(* IEC 61131-3 sources: test/Class/HmiComPortCan, 1 file *)

(* ---- HmiComPortCan.st ---- *)
(*!
<Class
	Name               = "HmiComPortCan"
	Revision           = "0.14"
	RealtimeTask       = "false"
	CyclicTask         = "false"
	BackgroundTask     = "false"
	Sigmatek           = "true"
	OSInterface        = "false"
	HighPriority       = "false"
	Automatic          = "false"
	UpdateMode         = "Prescan"
	SharedCommandTable = "true"
	Objectsize         = "(490,120)">
	<Channels>
		<Client Name="CanInterface" Required="true" Internal="false" DefValue="1"/>
		<Client Name="CanNodeDisplay" Required="true" Internal="false" DefValue="1"/>
		<Client Name="CanRxMsgID" Required="true" Internal="false" DefValue="16#40"/>
		<Client Name="CanSend" Required="true" Internal="true"/>
		<Client Name="CanTxMsgID" Required="true" Internal="false" DefValue="16#20"/>
		<Client Name="CoCanLib" Required="false" Internal="false"/>
	</Channels>
	<RevDoku>
		<Owner Company="sigmatek" Author="kolott"/>
		<Dokumentation Revision="0.14" Date="2015-06-11" Author="hoechr1" Company="sigmatek" Description="SA31241: inserted client for communication over hardware modules"/>
		<Dokumentation Revision="0.13" Date="2015-03-16" Author="kolott" Company="sigmatek" Description="SA30531: new Clients CanRxMsgID and CanTxMsgID"/>
		<Dokumentation Revision="0.12" Date="2014-11-27" Author="kolott" Company="sigmatek" Description="code reduced to can-connection"/>
		<Dokumentation Revision="0.11" Date="2014-08-28" Author="kolott" Company="sigmatek" Description="function &quot;UserCall&quot; added, extended timeout at flashkill &#13;&#10;retry implemented at method SendFile()"/>
		<Dokumentation Revision="0.10" Date="2014-06-13" Author="kolott" Company="sigmatek" Description="attribut &quot;virtual global&quot; added to method SendData()"/>
		<Dokumentation Revision="0.9" Date="2014-05-14" Author="kolott" Company="sigmatek" Description="evaluate retcode of method UpdateData()"/>
		<Dokumentation Revision="0.8" Date="2014-04-24" Author="kolott" Company="sigmatek" Description="new Method SendRestartSetup()"/>
		<Dokumentation Revision="0.7" Date="2014-04-02" Author="kolott" Company="sigmatek" Description="ErrorCnt will count on tx error as well"/>
		<Dokumentation Revision="0.6" Date="2014-03-04" Author="kolott" Company="sigmatek" Description="new Method GetNode()"/>
		<Dokumentation Revision="0.5" Date="2014-02-21" Author="kolott" Company="sigmatek" Description="new Method: GetHwVersion(), GetSwVersion()"/>
		<Dokumentation Revision="0.4" Date="2014-02-13" Author="kolott" Company="sigmatek" Description="innovation"/>
		<Dokumentation Revision="0.3" Date="2014-02-12" Author="kolott" Company="sigmatek" Description="new command LastUsage of HMI implemented"/>
		<Dokumentation Revision="0.2" Date="2014-01-29" Author="kolott" Company="sigmatek" Description="innovation: speed"/>
		<Dokumentation Revision="0.1" Date="2014-01-16" Author="kolott" Company="sigmatek" Description="method SendTrendValue added"/>
	</RevDoku>
	<Network Name="HmiComPortCan">
		<!-- List of Components in this network -->
		<Components>
			<Object
				Name       = "_base"
				Class      = "HmiComPort"
				Position   = "(218,120)"
				Visualized = "false">
				<Channels>
					<Server Name="ClassSvr"/>
					<Server Name="ErrorCnt"/>
					<Server Name="RetryCnt"/>
					<Server Name="RxData"/>
					<Server Name="TxData"/>
					<Client Name="CoSys"/>
					<Client Name="StdLib"/>
				</Channels>
			</Object>
			<Object
				Name       = "CanSend"
				Class      = "HmiCanSendReceive"
				Position   = "(210,510)"
				Visualized = "false">
				<Channels>
					<Server Name="ClassSvr"/>
					<Server Name="ErrorCnt"/>
					<Server Name="RxPack"/>
					<Server Name="TxPack"/>
					<Server Name="TxRetry"/>
					<Client Name="CanInterface" Value="1"/>
					<Client Name="CanNodeDisplay" Value="1"/>
					<Client Name="CanRxMsgID" Value="16#40"/>
					<Client Name="CanTxMsgID" Value="16#20"/>
					<Client Name="CoCan"/>
					<Client Name="CoCanLib"/>
					<Client Name="CoSys"/>
				</Channels>
			</Object>
		</Components>
		<Comments>
		</Comments>
		<!-- List of Connections in this network -->
		<Connections>
			<Connection Source="this.ClassSvr" Destination="_base.ClassSvr" Vertices="(690,210),(518,210),"/>
			<Connection Source="this.CanSend" Destination="CanSend.ClassSvr"/>
			<Connection Source="CanSend.CanNodeDisplay" Destination="this.CanNodeDisplay" Vertices="(210,600),(38,510),"/>
			<Connection Source="CanSend.CanInterface" Destination="this.CanInterface" Vertices="(210,660),(38,570),"/>
			<Connection Source="this.RxData" Destination="_base.RxData" Vertices="(690,270),(518,270),"/>
			<Connection Source="this.TxData" Destination="_base.TxData" Vertices="(690,330),(518,330),"/>
			<Connection Source="this.ErrorCnt" Destination="_base.ErrorCnt" Vertices="(690,390),(518,390),"/>
			<Connection Source="this.RetryCnt" Destination="_base.RetryCnt" Vertices="(690,450),(518,450),"/>
			<Connection Source="CanSend.CanRxMsgID" Destination="this.CanRxMsgID" Vertices="(210,720),(38,630),"/>
			<Connection Source="CanSend.CanTxMsgID" Destination="this.CanTxMsgID" Vertices="(210,780),(38,690),"/>
			<Connection Source="CanSend.CoCanLib" Destination="this.CoCanLib" Vertices="(210,960),(38,750),"/>
		</Connections>
		<!-- Headerfiles -->
		<Options>
		</Options>
	</Network>
</Class>
*)
#pragma using HmiComPort

HmiComPortCan : CLASS
: HmiComPort
  //Servers:
  //Clients:
	CanNodeDisplay 	: CltCh_DINT;
	CanInterface 	: CltCh_DINT;
	CanSend 	: CltChCmd_HmiCanSendReceive;
	CanRxMsgID 	: CltCh_DINT;
	CanTxMsgID 	: CltCh_DINT;
	CoCanLib 	: CltChCmd__CanLib;
  //Variables:
		RxCrc 	: UDINT;
		Crc 	: UDINT;
  //Functions:

	FUNCTION VIRTUAL GLOBAL Start
		VAR_INPUT
			pthis 	: ^void;
		END_VAR;

	FUNCTION VIRTUAL GLOBAL GetNode
		VAR_OUTPUT
			retcode 	: UDINT;
		END_VAR;

	FUNCTION VIRTUAL SendDataIntern
		VAR_INPUT
			src 	: ^void;
			size 	: UDINT;
		END_VAR
		VAR_OUTPUT
			retcode 	: BOOL;
		END_VAR;
				//! <Function Comment="Get timeout in milliseconds to wait for rx-data" Name="GetRxTimeout"/>
	FUNCTION VIRTUAL GetRxTimeout
		VAR_INPUT
			index 	: TRxTimeout;
		END_VAR
		VAR_OUTPUT
			retcode 	: UDINT;
		END_VAR;

	FUNCTION GLOBAL RxCallback
		VAR_INPUT
			pthis 	: ^HmiComPortCan;
			pdata 	: ^USINT;
			size 	: UDINT;
		END_VAR;
  //Tables:
	FUNCTION @STD
		VAR_OUTPUT
			ret_code	: CONFSTATES;
		END_VAR;
	FUNCTION GLOBAL TAB @CT_;
END_CLASS;

#pragma using HmiCanSendReceive
#pragma usingLtd _CanLib

FUNCTION VIRTUAL GLOBAL HmiComPortCan::Start
	VAR_INPUT
		pthis 	: ^void;
	END_VAR

  HmiComPort::Start(pthis);
  CanSend.Start(#RxCallback(), this);
  RetryNo := 2;  // 2 retry after first fail

END_FUNCTION

FUNCTION GLOBAL HmiComPortCan::RxCallback
	VAR_INPUT
		pthis 	: ^HmiComPortCan;
		pdata 	: ^USINT;
		size 	: UDINT;
	END_VAR

  this := pthis;
  RecieveData(pdata, size);

END_FUNCTION

FUNCTION VIRTUAL GLOBAL HmiComPortCan::GetNode
	VAR_OUTPUT
		retcode 	: UDINT;
	END_VAR

  retcode := to_udint(CanNodeDisplay);

END_FUNCTION

FUNCTION VIRTUAL HmiComPortCan::GetRxTimeout
	VAR_INPUT
		index 	: TRxTimeout;
	END_VAR
	VAR_OUTPUT
		retcode 	: UDINT;
	END_VAR

  retcode := HmiComPort::GetRxTimeout(index);
  case index of
    RxDelayStandard   : retcode :=   150;
    RxDelayFlashWrite : retcode := 40000;
    RxDelayFlashKill  : retcode :=  3000;
  end_case;

END_FUNCTION

FUNCTION VIRTUAL HmiComPortCan::SendDataIntern
	VAR_INPUT
		src 	: ^void;
		size 	: UDINT;
	END_VAR
	VAR_OUTPUT
		retcode 	: BOOL;
	END_VAR

  //  WaitBusy();
  retcode := CanSend.SendData(src, size);

END_FUNCTION
